// TIA Portal V20 export
TYPE "IO_Device_Functinal_Test_Rework"
   STRUCT
      Life_Trigger_PLC_Functional_Test_Rework : Bool;
      Star_Test_PLC_Functional_Test_Rework : Bool;
      Button_PLC_Functional_Test_Rework : Bool;
      Electrical_Current_Test_Approved_PLC_Functional_Test_Rework : Bool;
      Visual_Test_Approved_PLC_Functional_Test_Rework : Bool;
      Electrical_Current_Read_PLC_Functional_Test_Rework : UInt;
   END_STRUCT;
END_TYPE
